Staubli VAL3: lookForInstr.pgx

program lookForInstr(string& x_sItemToFind[] (dimensions=1), string& x_sItem[] (dimensions=1), bool& x_bFound[] (dimensions=1))
  local num l_nPos
  local bool l_bContinue
begin
  // init
  x_bFound=false
  // look for deep scan or not
  if size(x_sItemToFind)>1
    // find which instruction is
    l_nPos=find(x_sItem,x_sItemToFind)
    if l_nPos!=-1
      // look if the find give a correct answer
      // look before and after
      if l_nPos==0 or (asc(x_sItem,l_nPos-1)<65 or asc(x_sItem,l_nPos-1)>90)
        // continue
        /// OK check for the instruction now
        l_nPos=find(x_sItem,x_sItemToFind[1])
        // look if before is empty
        if asc(x_sItem,l_nPos-1)==32 and l_nPos!=-1
          x_bFound=true
        endIf
      endIf
    endIf
  else
    // NORMAL SEARCH
    if x_sItem==x_sItemToFind
      x_bFound=true
    endIf
  endIf
end
